(* Logix 5000 project; controller Std_Conveyors Emulate 5570 rev 32.11; software revision 32.01 *)

TASK MainTask (continuous, watchdog 500 ms) : MainProgram

MODULES
   Local : Emulate 5570 (ICP 0, rev 32.11)
      Ethernet : vendor 1 type 12 code 20 (ICP 1, Ethernet 192.168.1.13, rev 2.1)
END_MODULES

ADD_ON_INSTRUCTION AOI_Conveyors   (* revision 1.0, vendor Mirs-AG180725 *)
VAR_INPUT
   InMode : INT; {required}   // 1 for auto mode 2 for manual mode 3 for service mode
END_VAR
VAR_OUTPUT
   OutMode : DINT; {access Read Only, visible}   // 1 for auto mode 2 for manual mode 3 for service mode
   Out_Mapping : INT; {access Read Only, visible}
        .0   // Auto Mode
        .1   // Manual Mode
        .2   // Service Mode
        .3   // Ready to Receive
        .4   // Sensor Config Error
        .5   // Feedback auto mode
        .6   // feedback manual mode
        .7   // feedback service mode
END_VAR
VAR_INPUT
   InSensorConfig : INT; {required}
   IN_POSMapping : DINT; {required}
   IN_PREMapping : DINT; {required}
   IN_TransferMode : INT; {required}
   IN_SetWaitTimeReceived : DINT; {required}
   IN_SetWaitTimeDelivering : DINT; {required}
   IN_SetDelayReceiving : DINT; {required}
   IN_SetDelayDelivering : DINT; {required}
   IN_ESGlobal : BOOL; {required}
   IN_ESLocal : BOOL; {access None, required}
   IN_SetTransferMode : INT; {required}
   IN_BlockConveyors : BOOL; {required}
   In_ReleaseProduct : BOOL;
END_VAR
VAR_OUTPUT
   Running : BOOL; {visible}
   AutoMode : BOOL; {visible}
   ManualMode : BOOL; {visible}
   ServiceMode : BOOL; {visible}
   Out_StartMotor : BOOL; {visible}
   WithProduct : BOOL; {visible}
   Ocupied : BOOL; {visible}
   ReadyToReceive : BOOL; {visible}
   Delivering : BOOL; {visible}
   Receiving : BOOL; {visible}
   Blocked : BOOL; {visible}
   Starving : BOOL; {visible}
   TimeoutReceiving : BOOL; {visible}
   TimeOutDelivering : BOOL; {visible}
   Fault : BOOL; {visible}
END_VAR
VAR_INPUT
   In_Sensor1 : BOOL;   // 0 free 1 presence
   In_Sensor2 : BOOL;   // 0 free 1 presence
   StartConveyor : BOOL;
   StopConveyors : BOOL;
END_VAR
VAR
   UseOnlyExitLogic : BOOL;
   UseOnlyOcuppiedLogic : BOOL;
   WaitTimeReceived : TIMER; {access None}
   CheckingStatus : BOOL; {access None}
   aux_Init : TIMER := (PRE := 5000); {access None}
   SetInitTime : DINT; {access None}
END_VAR

ROUTINE Logic   (* ladder *)
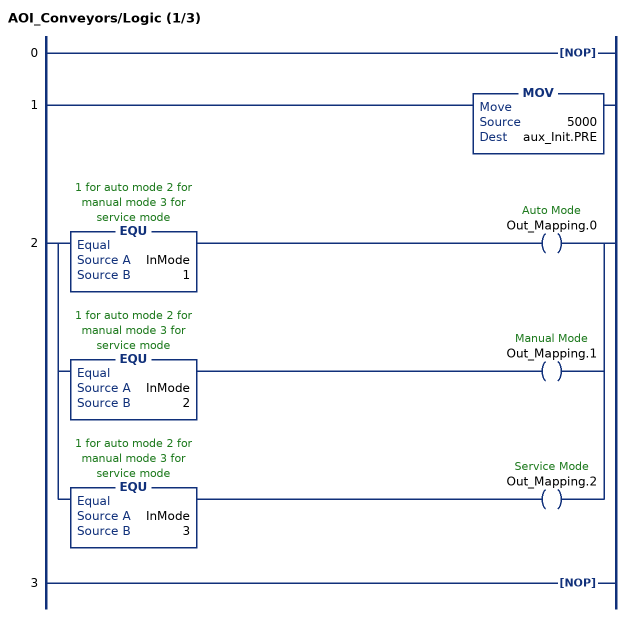
   0: NOP();
   1: MOV(5000,aux_Init.PRE);
   2: [EQU(InMode,1) OTE(Out_Mapping.0) ,EQU(InMode,2) OTE(Out_Mapping.1) ,EQU(InMode,3) OTE(Out_Mapping.2) ];
   3: NOP();
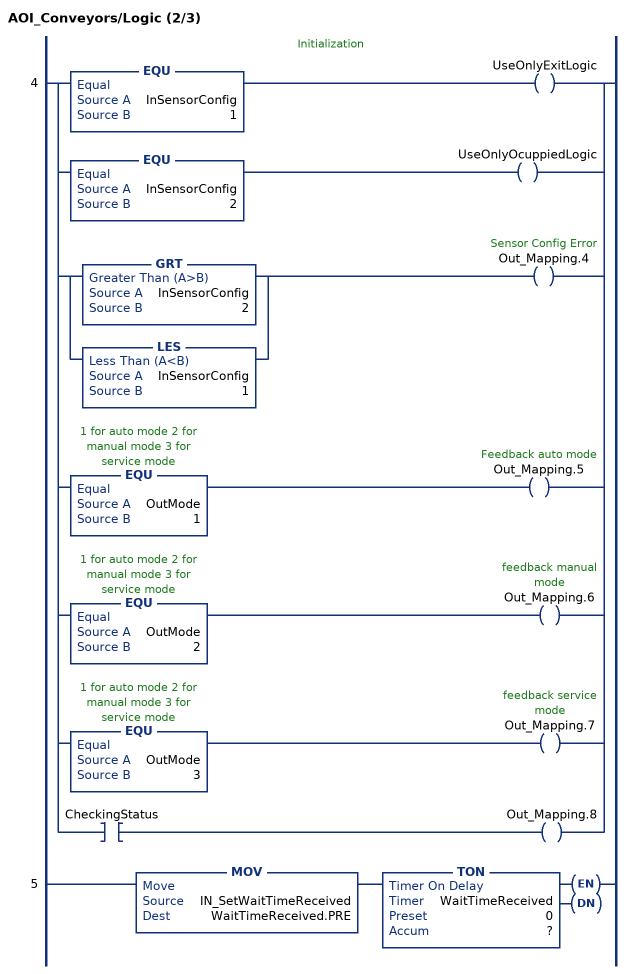
   // Initialization
   4: [EQU(InSensorConfig,1) OTE(UseOnlyExitLogic) ,EQU(InSensorConfig,2) OTE(UseOnlyOcuppiedLogic) ,[GRT(InSensorConfig,2) ,LES(InSensorConfig,1) ] OTE(Out_Mapping.4) ,EQU(OutMode,1) OTE(Out_Mapping.5) ,EQU(OutMode,2) OTE(Out_Mapping.6) ,EQU(OutMode,3) OTE(Out_Mapping.7) ,XIC(CheckingStatus) OTE(Out_Mapping.8) ];
   5: MOV(IN_SetWaitTimeReceived,WaitTimeReceived.PRE)TON(WaitTimeReceived,?,?);
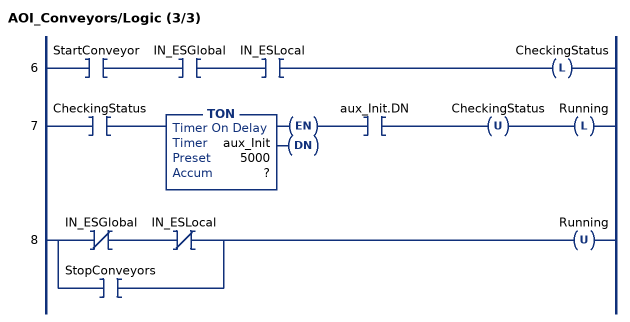
   6: XIC(StartConveyor)XIC(IN_ESGlobal)XIC(IN_ESLocal)OTL(CheckingStatus);
   7: XIC(CheckingStatus)TON(aux_Init,?,?)XIC(aux_Init.DN)OTU(CheckingStatus)OTL(Running);
   8: [XIO(IN_ESGlobal) XIO(IN_ESLocal) ,XIC(StopConveyors) ]OTU(Running);
END_ROUTINE
END_ADD_ON_INSTRUCTION

VAR_GLOBAL   (* controller tags *)
   _auxRbtBlockConveyor : BOOL;
   _EHMI_I_EmitirCaja : ALIAS FOR _EHMI_I_MAP[0].0;
   _EHMI_I_MAP : INT[200];
   _EHMI_O_MAP : INT[200];
   _glbBlockConveyors : BOOL;
   _ModeInfeed : DINT := 1;
   _ModeOutfeed : DINT := 3;
   _ModeRunning : INT := 1;
   _ModeTransfer : DINT := 2;
   _RbtBlockConveyor : BOOL;
   _safetySys : BOOL := 1;
   _safetySysLocalCv : BOOL := 1;
   _Sensor1_T1 : BOOL;
   _Sensor1_T2 : BOOL;
   _Sensor1_T3 : BOOL;
   _Sensor1_T4 : BOOL;
   _Sensor2_T1 : BOOL;
   _Sensor2_T2 : BOOL;
   _Sensor2_T3 : BOOL;
   _Sensor2_T4 : BOOL;
   _SensorConfig : DINT := 1;
   _SetDelayDelivering : DINT := 2000;
   _SetDelayReceiving : DINT := 2000;
   _SetWaitTimeDelivering : DINT := 2000;
   _SetWaitTimeReceiving : DINT := 2000;
   _SynOSeq : DINT := 1;   // 1 Synchronous 2 sequential
   AuxBlockConveyor : BOOL;
   BOOL_IN_0 : BOOL;
   BOOL_IN_1 : BOOL;
   BOOL_IN_5 : BOOL := 1;
   BOOL_OUT_0 : BOOL;
   BOOL_OUT_1 : BOOL;
   Conveyor1 : AOI_Conveyors := (InMode := 1, Out_Mapping := 1, InSensorConfig := 1, IN_POSMapping := 1, IN_PREMapping := 1, IN_TransferMode := 1, IN_SetWaitTimeReceived := 2000, IN_SetWaitTimeDelivering := 2000, IN_SetDelayReceiving := 2000, IN_SetDelayDelivering := 2000, IN_ESGlobal := 1, IN_ESLocal := 1, IN_SetTransferMode := 1);
   Conveyor2 : AOI_Conveyors := (InMode := 1, Out_Mapping := 1, InSensorConfig := 1, IN_POSMapping := 1, IN_PREMapping := 1, IN_TransferMode := 2, IN_SetWaitTimeReceived := 2000, IN_SetWaitTimeDelivering := 2000, IN_SetDelayReceiving := 2000, IN_SetDelayDelivering := 2000, IN_ESGlobal := 1, IN_ESLocal := 1, IN_SetTransferMode := 1);
   conveyor3 : AOI_Conveyors := (InMode := 1, Out_Mapping := 1, InSensorConfig := 1, IN_POSMapping := 1, IN_PREMapping := 1, IN_TransferMode := 3, IN_SetWaitTimeReceived := 2000, IN_SetWaitTimeDelivering := 2000, IN_SetDelayReceiving := 2000, IN_SetDelayDelivering := 2000, IN_ESGlobal := 1, IN_ESLocal := 1, IN_SetTransferMode := 1);
   conveyor4 : AOI_Conveyors := (InMode := 1, Out_Mapping := 1, InSensorConfig := 1, IN_POSMapping := 1, IN_PREMapping := 1, IN_TransferMode := 3, IN_SetWaitTimeReceived := 2000, IN_SetWaitTimeDelivering := 2000, IN_SetDelayReceiving := 2000, IN_SetDelayDelivering := 2000, IN_ESGlobal := 1, IN_ESLocal := 1, IN_SetTransferMode := 1);
   motor1 : BOOL;
   motor2 : BOOL;
   motor3 : BOOL;
   motor4 : BOOL;
   plsReleaseCv : BOOL;
   ReleaseCVByRbt : BOOL;
   Sim_I_btn_Emitir : ALIAS FOR BOOL_IN_1;
   Sim_I_sensor_Remover : ALIAS FOR BOOL_IN_0;
   Sim_O_Emitir : ALIAS FOR BOOL_OUT_1;
   Sim_O_Remover : ALIAS FOR BOOL_OUT_0;
   time2 : TIMER;
END_VAR

PROGRAM MainProgram   (* main routine MainRoutine *)

ROUTINE _ConveyorsLogic   (* ladder *)
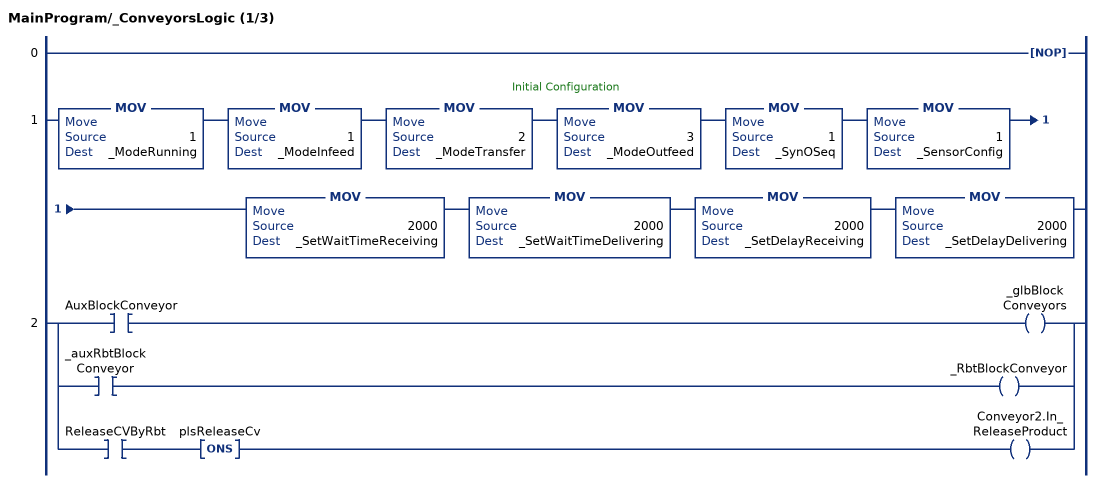
   0: NOP();
   // Initial Configuration
   1: MOV(1,_ModeRunning)MOV(1,_ModeInfeed)MOV(2,_ModeTransfer)MOV(3,_ModeOutfeed)MOV(1,_SynOSeq)MOV(1,_SensorConfig)MOV(2000,_SetWaitTimeReceiving)MOV(2000,_SetWaitTimeDelivering)MOV(2000,_SetDelayReceiving)MOV(2000,_SetDelayDelivering);
   2: [XIC(AuxBlockConveyor) OTE(_glbBlockConveyors) ,XIC(_auxRbtBlockConveyor) OTE(_RbtBlockConveyor) ,XIC(ReleaseCVByRbt) ONS(plsReleaseCv) OTE(Conveyor2.In_ReleaseProduct) ];
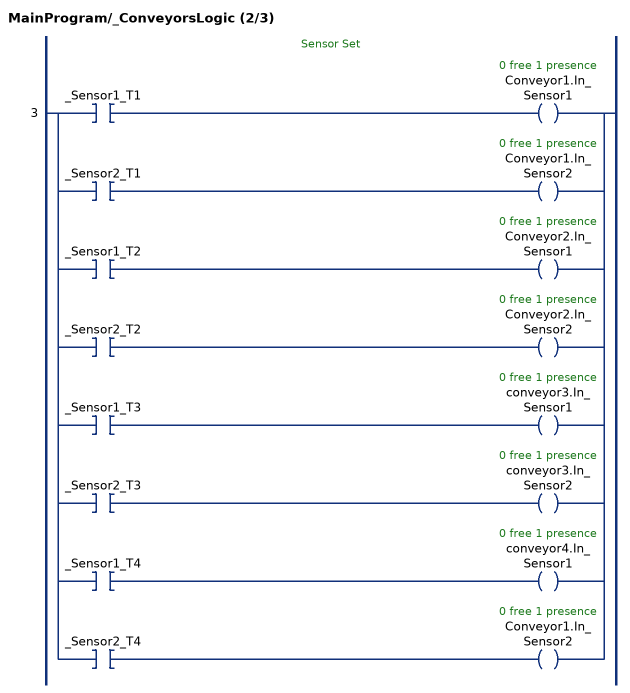
   // Sensor Set
   3: [XIC(_Sensor1_T1) OTE(Conveyor1.In_Sensor1) ,XIC(_Sensor2_T1) OTE(Conveyor1.In_Sensor2) ,XIC(_Sensor1_T2) OTE(Conveyor2.In_Sensor1) ,XIC(_Sensor2_T2) OTE(Conveyor2.In_Sensor2) ,XIC(_Sensor1_T3) OTE(conveyor3.In_Sensor1) ,XIC(_Sensor2_T3) OTE(conveyor3.In_Sensor2) ,XIC(_Sensor1_T4) OTE(conveyor4.In_Sensor1) ,XIC(_Sensor2_T4) OTE(Conveyor1.In_Sensor2) ];
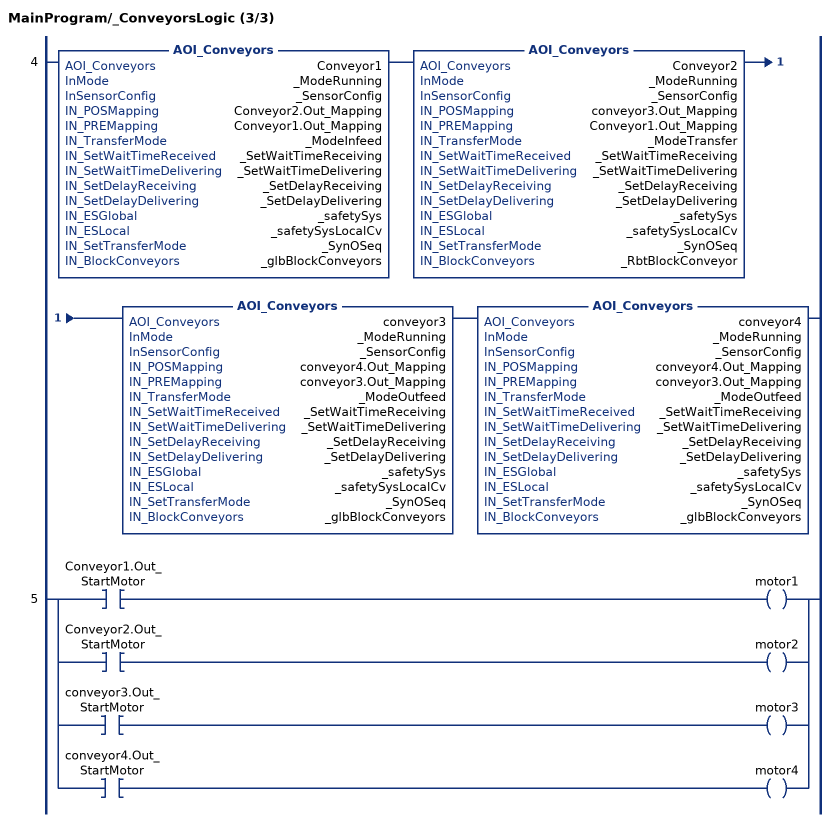
   4: AOI_Conveyors(Conveyor1,_ModeRunning,_SensorConfig,Conveyor2.Out_Mapping,Conveyor1.Out_Mapping,_ModeInfeed,_SetWaitTimeReceiving,_SetWaitTimeDelivering,_SetDelayReceiving,_SetDelayDelivering,_safetySys,_safetySysLocalCv,_SynOSeq,_glbBlockConveyors)AOI_Conveyors(Conveyor2,_ModeRunning,_SensorConfig,conveyor3.Out_Mapping,Conveyor1.Out_Mapping,_ModeTransfer,_SetWaitTimeReceiving,_SetWaitTimeDelivering,_SetDelayReceiving,_SetDelayDelivering,_safetySys,_safetySysLocalCv,_SynOSeq,_RbtBlockConveyor)AOI_Conveyors(conveyor3,_ModeRunning,_SensorConfig,conveyor4.Out_Mapping,conveyor3.Out_Mapping,_ModeOutfeed,_SetWaitTimeReceiving,_SetWaitTimeDelivering,_SetDelayReceiving,_SetDelayDelivering,_safetySys,_safetySysLocalCv,_SynOSeq,_glbBlockConveyors)AOI_Conveyors(conveyor4,_ModeRunning,_SensorConfig,conveyor4.Out_Mapping,conveyor3.Out_Mapping,_ModeOutfeed,_SetWaitTimeReceiving,_SetWaitTimeDelivering,_SetDelayReceiving,_SetDelayDelivering,_safetySys,_safetySysLocalCv,_SynOSeq,_glbBlockConveyors);
   5: [XIC(Conveyor1.Out_StartMotor) OTE(motor1) ,XIC(Conveyor2.Out_StartMotor) OTE(motor2) ,XIC(conveyor3.Out_StartMotor) OTE(motor3) ,XIC(conveyor4.Out_StartMotor) OTE(motor4) ];
END_ROUTINE

ROUTINE MainRoutine   (* ladder *)
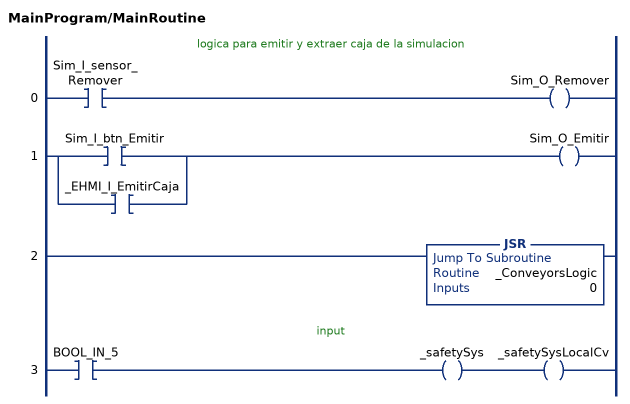
   // logica para emitir y extraer caja de la simulacion
   0: XIC(Sim_I_sensor_Remover)OTE(Sim_O_Remover);
   1: [XIC(Sim_I_btn_Emitir) ,XIC(_EHMI_I_EmitirCaja) ]OTE(Sim_O_Emitir);
   2: JSR(_ConveyorsLogic,0);
   // input
   3: XIC(BOOL_IN_5)OTE(_safetySys)OTE(_safetySysLocalCv);
END_ROUTINE
END_PROGRAM
